FUNCTION_BLOCK FB_RCC_SM
VAR_IN_OUT
    stRCC_VRC_01 : ST_VRC;
    stRCC_VRC_02 : ST_VRC;
    stRCC_VRC_03 : ST_VRC;
    stRCC_VRC_04 : ST_VRC;
    stRCC_GCP_01 : ST_VG;

    TInterval : TIME; // Time in between cycles
    T1 : TIME;
    T2 : TIME;
    T3 : TIME;
    T4 : TIME;

    bRunClean : BOOL;
    bClearError : BOOL;
    bError : BOOL;
    bStop : BOOL;
    bStartCycle : BOOL;
    bRunning : BOOL;
    tTimerRBV : STRING;

    RCC_GCP_01_INTERLOCK_SETPOINT : REAL;
    xSystemOverrideMode_RCC : BOOL;
    eCurrentState : INT;
    sLogMessage : T_MaxString;

    RCC_VRC_01_OPEN_OK : BOOL;
    RCC_VRC_02_OPEN_OK : BOOL;
    RCC_VRC_03_OPEN_OK : BOOL;
    RCC_VRC_04_OPEN_OK : BOOL;
END_VAR
VAR
    RCC_GCP_ILK_CONV : REAL;
    tTimer1 : TON;
END_VAR

RCC_GCP_ILK_CONV := RCC_GCP_01_INTERLOCK_SETPOINT * 1E2; // Convert to Torr
tTimerRBV := TIME_TO_STRING(tTimer1.ET);

(* Valve can open only when CRIX-RCC-VRC-02 and 03 are closed*)
RCC_VRC_01_OPEN_OK := ( stRCC_VRC_02.i_xClsLS AND NOT stRCC_VRC_02.q_xOPN_DO ) AND
                                    ( stRCC_VRC_03.i_xClsLS AND NOT stRCC_VRC_03.q_xOPN_DO ) ;

(* Valve can open only when CRIX-RCC-VRC-01 and 04 are closed*)
RCC_VRC_02_OPEN_OK := ( stRCC_VRC_01.i_xClsLS AND NOT stRCC_VRC_01.q_xOPN_DO ) AND
                                    ( stRCC_VRC_04.i_xClsLS AND NOT stRCC_VRC_04.q_xOPN_DO );

(* Valve can open only when CRIX-RCC-GCP-01 reading < setpoint Torr and CRIX-RCC-VRC-01 and 04 are closed*)
RCC_VRC_03_OPEN_OK := (stRCC_GCP_01.rPRESS < RCC_GCP_ILK_CONV AND stRCC_GCP_01.xPRESS_OK ) AND
                                 ( stRCC_VRC_01.i_xClsLS AND NOT stRCC_VRC_01.q_xOPN_DO ) AND
                                              ( stRCC_VRC_04.i_xClsLS AND NOT stRCC_VRC_04.q_xOPN_DO );


(* Valve can open only when CRIX-RCC-VRC-02 and 03 are closed*)
RCC_VRC_04_OPEN_OK := ( stRCC_VRC_02.i_xClsLS AND NOT stRCC_VRC_02.q_xOPN_DO ) AND
                                      ( stRCC_VRC_03.i_xClsLS AND NOT stRCC_VRC_03.q_xOPN_DO ) ;


IF bStop THEN
    eCurrentState:= E_RCC_STATES.INIT;
    bStartCycle := FALSE;
END_IF

 CASE eCurrentState OF
    E_RCC_STATES.ERROR: // SOMETHING WENT WRONG
        bRunning := FALSE;
        stRCC_VRC_01.pv_xOPN_SW := FALSE;
        stRCC_VRC_02.pv_xOPN_SW := FALSE;
        stRCC_VRC_03.pv_xOPN_SW := FALSE;
        stRCC_VRC_04.pv_xOPN_SW := FALSE;

        IF bClearError THEN
            eCurrentState := E_RCC_STATES.IDLE;
            bError := FALSE;
            bClearError:= FALSE;
        END_IF

    E_RCC_STATES.IDLE: // -1
        sLogMessage := 'IDLE';
        bRunning := FALSE;
        IF bStartCycle THEN
            tTimer1(IN:=FALSE); // RESTART TIMER
            eCurrentState := E_RCC_STATES.INIT;
            bRunning := TRUE;
        END_IF

    E_RCC_STATES.INIT: // 0
        sLogMessage := 'WAITING FOR CYCLE TO START';
        stRCC_VRC_01.pv_xOPN_SW := FALSE;
        stRCC_VRC_02.pv_xOPN_SW := FALSE;
        stRCC_VRC_03.pv_xOPN_SW := FALSE;
        stRCC_VRC_04.pv_xOPN_SW := FALSE;
        tTimer1(IN:=TRUE, PT:=TInterval);

        IF tTimer1.Q THEN
            eCurrentState:= E_RCC_STATES.OPEN_VRC_02_FOR_T1;
            tTimer1(IN:=FALSE); // RESTART TIMER
        END_IF

        IF bStop THEN
            eCurrentState:= E_RCC_STATES.IDLE;
            bStop := FALSE;
        END_IF

    E_RCC_STATES.OPEN_VRC_02_FOR_T1: // OPEN 1
        sLogMessage := 'OPEN VAVLE 2 FOR T1 SECONDS';
        tTimer1(IN:=TRUE, PT:=T1);
        stRCC_VRC_02.pv_xOPN_SW := TRUE;

        IF tTimer1.Q THEN
            eCurrentState := E_RCC_STATES.DRAIN;
            tTimer1(IN:=FALSE); // RESTART TIMER
        END_IF

     E_RCC_STATES.DRAIN:	// DRAIN_1 2
        // THIS MIGHT CAUSE THE RCC TO STALL IF THIS CONDITION IS NEVER MET
        sLogMessage := 'DRAINING';
        IF (NOT stRCC_GCP_01.xPRESS_OK) THEN
            eCurrentState := E_RCC_STATES.ERROR;
            bError := TRUE;
        END_IF

        IF RCC_VRC_03_OPEN_OK THEN
            IF bRunClean THEN stRCC_VRC_02.pv_xOPN_SW := FALSE; END_IF
            stRCC_VRC_03.pv_xOPN_SW := TRUE;
            eCurrentState := E_RCC_STATES.DRAIN_CHECK;
        END_IF

    E_RCC_STATES.DRAIN_CHECK:	// CHECK IF WE ARE DON DRAINING 3
        tTimer1(IN:=TRUE, PT:=T2);
        sLogMessage := 'OPEN VALVE 3 FOR T2 SECONDS';

        IF tTimer1.Q THEN
            eCurrentState := E_RCC_STATES.OPEN_VRC_01_FOR_T3;
            IF NOT RCC_VRC_03_OPEN_OK THEN eCurrentState := E_RCC_STATES.OPEN_VRC_02_FOR_T1; END_IF
             stRCC_VRC_03.pv_xOPN_SW := FALSE;
            IF NOT bRunClean THEN stRCC_VRC_02.pv_xOPN_SW := FALSE; END_IF
            tTimer1(IN:=FALSE); // RESTART TIMER
        END_IF

     E_RCC_STATES.OPEN_VRC_01_FOR_T3: // OPEN VRC_01 for T3 4
         sLogMessage := 'OPEN VALVE 1 FOR T3 SECONDS';
        tTimer1(IN:=TRUE, PT:=T3);
        stRCC_VRC_01.pv_xOPN_SW := TRUE;
        IF tTimer1.Q THEN
            eCurrentState := E_RCC_STATES.OPEN_VRC_04_FOR_T4;
            tTimer1(IN:=FALSE); // RESTART TIMER
        END_IF

     E_RCC_STATES.OPEN_VRC_04_FOR_T4: // OPEN VRC_04 for T4 5
         sLogMessage := 'OPEN VALVE 4 FOR T4 SECONDS';
        tTimer1(IN:=TRUE, PT:=T4);
        stRCC_VRC_04.pv_xOPN_SW := TRUE;
        IF tTimer1.Q THEN
            sLogMessage := 'CLOSING VALVE 1&4, RESTARTING CYCLE';
            eCurrentState := E_RCC_STATES.IDLE;
            stRCC_VRC_01.pv_xOPN_SW := FALSE;
            stRCC_VRC_04.pv_xOPN_SW := FALSE;
            tTimer1(IN:=FALSE); // RESTART TIMER
        END_IF


END_CASE

END_FUNCTION_BLOCK

(* stored: Version 1.1.0.1, ProductVersion 3.1.4024.12
   POU FB_RCC_SM: Id {47a0acf2-060b-4e55-9edc-089d8f8e62bc}, SpecialFunc None *)
